Staubli VAL3: sendTrajPtFAck.pgx

public program sendTrajPtFAck()
  local num l_nRetVal
begin
  // send message length (prefix)
  call sendData(siTcpIpMotion,rosTrajPtFAck.prefix.nData,nInConnFlag)
  // send message header (msg type, comm type, reply code)
  call sendData(siTcpIpMotion,rosTrajPtFAck.header.nData,nInConnFlag)
  call sendData(siTcpIpMotion,rosTrajPtFAck.body.nData,nInConnFlag)
end
